(* CODESYS project Logger.xml

Project tree, tasks and I/O mapping:
  function block Logger [LD]
*)

// Logger
FUNCTION_BLOCK Logger
VAR_INPUT
END_VAR
VAR_OUTPUT
END_VAR
VAR
	Reset: BOOL;
	
	TimeMakingIce: TIME;
	TimeMakingIceTimer: RTON;
	MakingIceTriggers: UINT;
	MakingIceTriggerCounter: CTU;
	HopperSensorFaults: UINT;
	HopperSensorFaultCounter: CTU;
	MakingIceFaults: UINT;
	MakingIceFaultCounter: CTU;
	
END_VAR

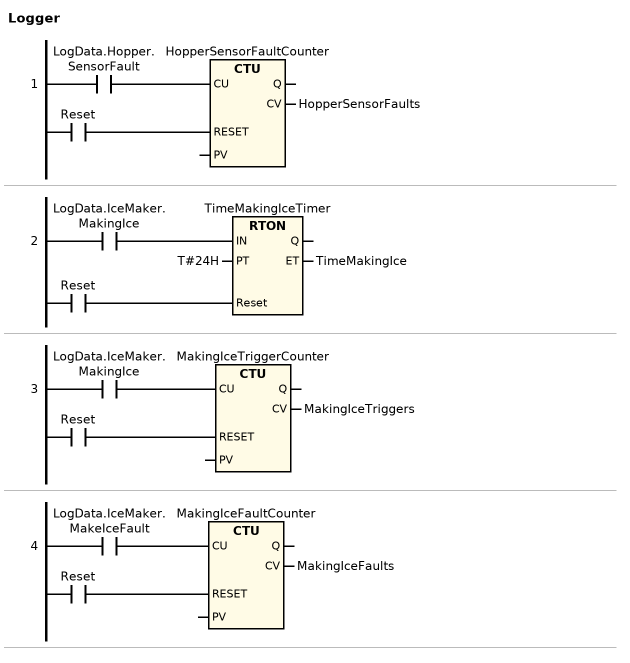
// NETWORK 1
HopperSensorFaultCounter(CU := LogData.Hopper.SensorFault, RESET := Reset, CV => HopperSensorFaults); // CTU

// NETWORK 2
TimeMakingIceTimer(IN := LogData.IceMaker.MakingIce, PT := T#24H, Reset := Reset, ET => TimeMakingIce); // RTON

// NETWORK 3
MakingIceTriggerCounter(CU := LogData.IceMaker.MakingIce, RESET := Reset, CV => MakingIceTriggers); // CTU

// NETWORK 4
MakingIceFaultCounter(CU := LogData.IceMaker.MakeIceFault, RESET := Reset, CV => MakingIceFaults); // CTU

END_FUNCTION_BLOCK
